FUNCTION_BLOCK E_TRAIN (* Generate of a finite train of events seperated by the time DT *)
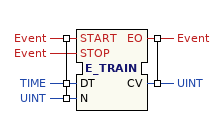
  EVENT_INPUT
    START WITH DT, N; (* Start event generation *)
    STOP; (* Stop event generation *)
  END_EVENT
  EVENT_OUTPUT
    EO WITH CV; (* Generated events *)
  END_EVENT
  VAR_INPUT
    DT : TIME; (* Time by which the events should be seperated *)
    N : UINT; (* Number of events to generate *)
  END_VAR
  VAR_OUTPUT
    CV : UINT; (* count of the current event: EO index (0..N-1) *)
  END_VAR
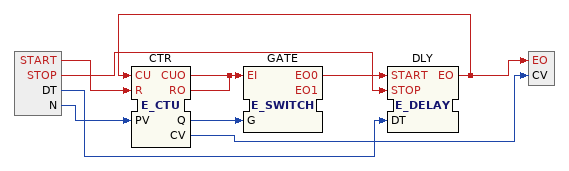
  FBS
    CTR : iec61499::events::E_CTU;
    GATE : iec61499::events::E_SWITCH;
    DLY : iec61499::events::E_DELAY;
  END_FBS
  EVENT_CONNECTIONS
    CTR.CUO TO GATE.EI;
    CTR.RO TO GATE.EI;
    START TO CTR.R;
    GATE.EO0 TO DLY.START;
    STOP TO DLY.STOP;
    DLY.EO TO EO;
    DLY.EO TO CTR.CU;
  END_CONNECTIONS
  DATA_CONNECTIONS
    N TO CTR.PV;
    CTR.CV TO CV;
    DT TO DLY.DT;
    CTR.Q TO GATE.G;
  END_CONNECTIONS
END_FUNCTION_BLOCK
